(* Logix 5000 project; controller DUNEW2PLC1 vendor 1 type 14 code 221 rev 33.11; software revision 33.00; part 6 of 7 *)
(* tags used below, declared in another part *)
   AbortQueue : BOOL;
   accel_xy : REAL;   // Tangential acceleration of the winding head in xy-plane
   ACTUATOR_POS : DINT;
   ALL_EOT_GOOD : BOOL;
   APA_IS_VERTICAL : BOOL;
   check_tension_stable : BOOL;   // Check if the tension is stable at the setpoint before moving the winding head
   CurIssued : BOOL;
   delay_mid_position : TIMER;
   ENABLE_ACTUATOR : BOOL;
   ERROR_CODE : DINT;
   FRAME_LOC_FT_BTM : BOOL;
   FRAME_LOC_FT_MID : BOOL;
   FRAME_LOC_FT_TOP : BOOL;
   FRAME_LOC_HD_BTM : BOOL;
   FRAME_LOC_HD_MID : BOOL;
   FRAME_LOC_HD_TOP : BOOL;
   gamma : REAL;
   INIT_DONE : BOOL;
   J : REAL;
   LATCH_ACTUATOR_HOMED : BOOL;
   LATCH_ACTUATOR_MID : BOOL;
   LATCH_ACTUATOR_TOP : BOOL;
   latching_in_progress : BOOL;
   MACHINE_SW_STAT : BOOL[32];
   MASTER_Z_GO : BOOL;
   MAX_TOLERABLE_Z : REAL;
   MCCD_X_Y_Axis1 : MOTION_INSTRUCTION;
   MOVE_TYPE : INT;   // 0 = No Move 1 = XY JOG 2 = XY Plane Move 3 = Z JOG 4 = Z Axis Move 5 = Toggle Latch Actuator 6 = Home the Latch Actuator
   NextIssued : BOOL;
   NEXTSTATE : DINT;
   no_apa_collision : BOOL;
   no_latch_collision : BOOL;
   no_supports_collision : BOOL;
   POSITION : REAL[1,2];
   QueueCount : DINT;
   speed_regulator_switch : BOOL;   // This is our "enable safe speed" switch, repurposed to switch the speed regulator
   STATE : DINT;   // CURRENT State Machine State
   STATE_FAULT_FLAGS : DINT;
   STATE_REQUEST : DINT;
   STATE_REQUEST_ACK : DINT;
   STATE_REQUEST_ID : DINT;
   STATE_REQUEST_RESULT : DINT;
   support_collision_window_bttm : BOOL;
   support_collision_window_mid : BOOL;
   support_collision_window_top : BOOL;
   tension : REAL;   // wire tension from load cell (N)
   TENSION_CONTROL_OK : BOOL;
   TENSION_ON_SWITCH : BOOL;
   tension_stable_timer : TIMER;
   v_0 : REAL;
   v_x_max : DINT;
   v_xyz : REAL;   // Velocity of winding head in xyz space
   v_y_max : DINT;
   X_axis : AXIS_CIP_DRIVE;
   X_POSITION : ALIAS FOR POSITION[0,0];
   X_XFER_OK : BOOL;   // If at the head, check head support arms. Same for foot
   X_Y : COORDINATE_SYSTEM;
   XY_ACCELERATION : REAL;   // Maximum positive acceleration for position move.
   XY_DECELERATION : REAL;   // Maximum negative acceleration for position move.
   xy_regulated_acceleration : REAL;
   xy_regulated_deceleration : REAL;
   XY_SPEED : REAL;   // Maximum velocity for position move.
   XY_SPEED_REQ : REAL;   // XY Requested speed copy of XY_Speed to be used for MCLM and MCCD in MoveXY
   xz : COORDINATE_SYSTEM;
   Y_axis : AXIS_CIP_DRIVE;
   Y_POSITION : ALIAS FOR POSITION[0,1];
   Y_XFER_OK : BOOL;
   Z_ACCELERATION : REAL;
   Z_axis : AXIS_CIP_DRIVE;
   Z_DECELLERATION : REAL;
   Z_EXTENDED : BOOL;
   Z_FIXED_LATCHED : BOOL;
   Z_FIXED_PRESENT : BOOL;
   Z_POSITION : REAL;
   Z_RETRACTED : BOOL;
   Z_SPEED : REAL;
   Z_STAGE_LATCHED : BOOL;
   Z_STAGE_PRESENT : BOOL;   // Winding head is on the Z-arm

PROGRAM state_14_hmi_stop   (* main routine main *)
VAR
   hmi_stop_entry_ob : BOOL;
   hmi_stop_entry_sb : BOOL;
   hmi_x_axis_stop : MOTION_INSTRUCTION := (FLAGS := 33554432);
   hmi_xy_stop : MOTION_INSTRUCTION := (FLAGS := 33554432);
   hmi_xz_stop : MOTION_INSTRUCTION := (FLAGS := 33554432);
   hmi_y_axis_stop : MOTION_INSTRUCTION := (FLAGS := 33554432);
   hmi_z_axis_stop : MOTION_INSTRUCTION := (FLAGS := 33554432);
   STATE14_IND : BOOL;
END_VAR

ROUTINE main   (* ladder *)
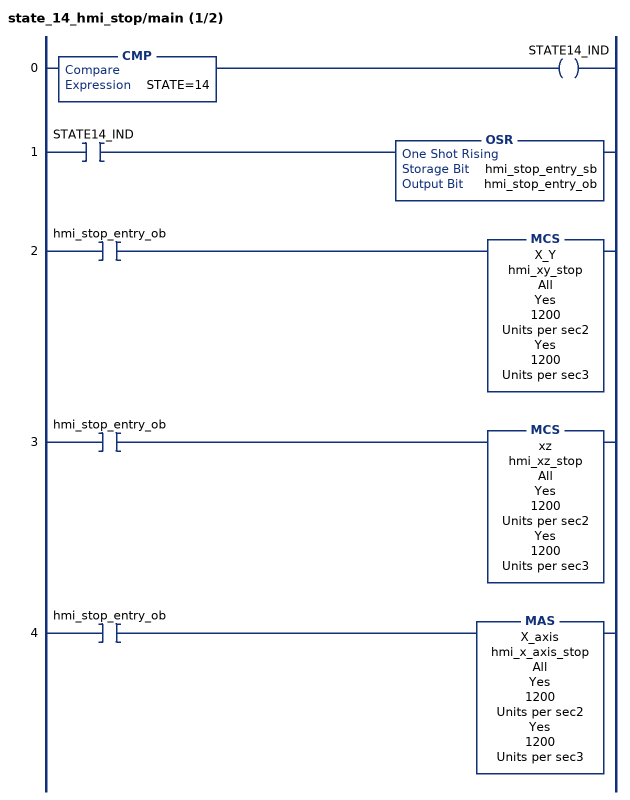
   0: CMP(STATE=14)OTE(STATE14_IND);
   1: XIC(STATE14_IND)OSR(hmi_stop_entry_sb,hmi_stop_entry_ob);
   2: XIC(hmi_stop_entry_ob)MCS(X_Y,hmi_xy_stop,All,Yes,1200,Units per sec2,Yes,1200,Units per sec3);
   3: XIC(hmi_stop_entry_ob)MCS(xz,hmi_xz_stop,All,Yes,1200,Units per sec2,Yes,1200,Units per sec3);
   4: XIC(hmi_stop_entry_ob)MAS(X_axis,hmi_x_axis_stop,All,Yes,1200,Units per sec2,Yes,1200,Units per sec3);
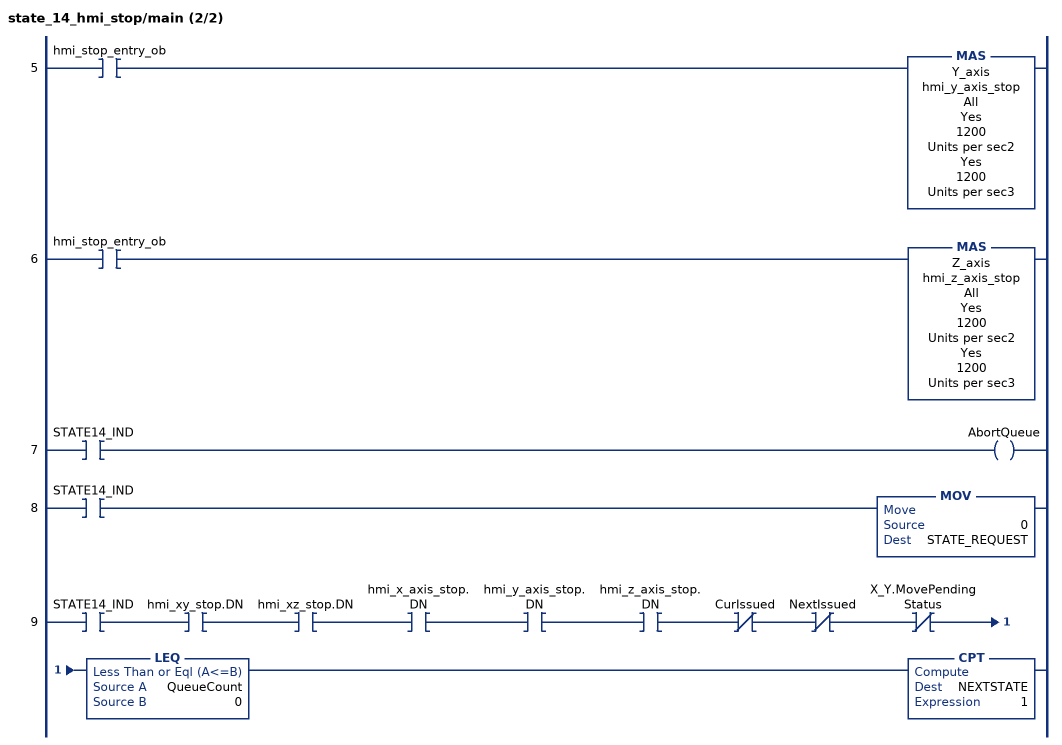
   5: XIC(hmi_stop_entry_ob)MAS(Y_axis,hmi_y_axis_stop,All,Yes,1200,Units per sec2,Yes,1200,Units per sec3);
   6: XIC(hmi_stop_entry_ob)MAS(Z_axis,hmi_z_axis_stop,All,Yes,1200,Units per sec2,Yes,1200,Units per sec3);
   7: XIC(STATE14_IND)OTE(AbortQueue);
   8: XIC(STATE14_IND)MOV(0,STATE_REQUEST);
   9: XIC(STATE14_IND)XIC(hmi_xy_stop.DN)XIC(hmi_xz_stop.DN)XIC(hmi_x_axis_stop.DN)XIC(hmi_y_axis_stop.DN)XIC(hmi_z_axis_stop.DN)XIO(CurIssued)XIO(NextIssued)XIO(X_Y.MovePendingStatus)LEQ(QueueCount,0)CPT(NEXTSTATE,1);
END_ROUTINE
END_PROGRAM

PROGRAM state_1_ready   (* main routine main *)
VAR
   STATE1_IND : BOOL; {access Read Only}
END_VAR

ROUTINE main   (* ladder *)
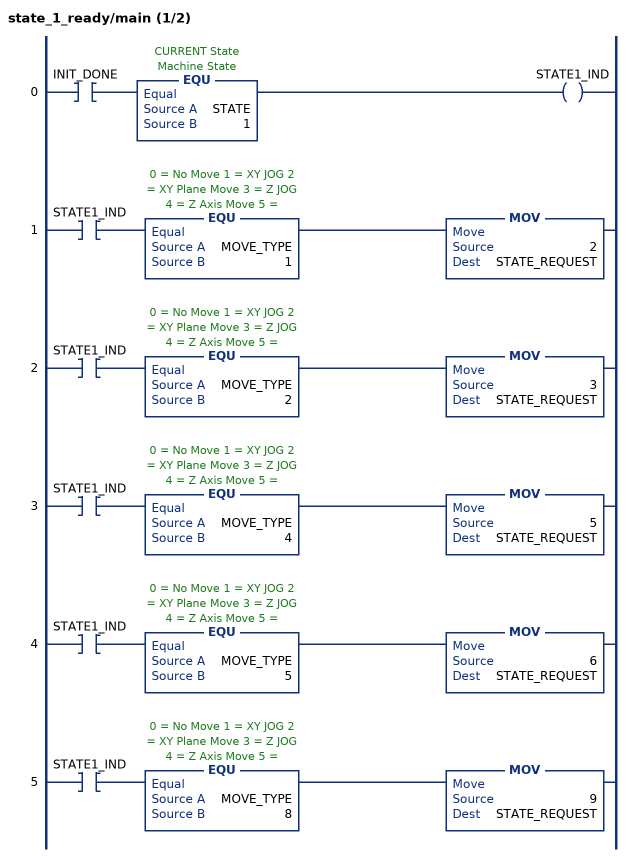
   0: XIC(INIT_DONE)EQU(STATE,1)OTE(STATE1_IND);
   1: XIC(STATE1_IND)EQU(MOVE_TYPE,1)MOV(2,STATE_REQUEST);
   2: XIC(STATE1_IND)EQU(MOVE_TYPE,2)MOV(3,STATE_REQUEST);
   3: XIC(STATE1_IND)EQU(MOVE_TYPE,4)MOV(5,STATE_REQUEST);
   4: XIC(STATE1_IND)EQU(MOVE_TYPE,5)MOV(6,STATE_REQUEST);
   5: XIC(STATE1_IND)EQU(MOVE_TYPE,8)MOV(9,STATE_REQUEST);
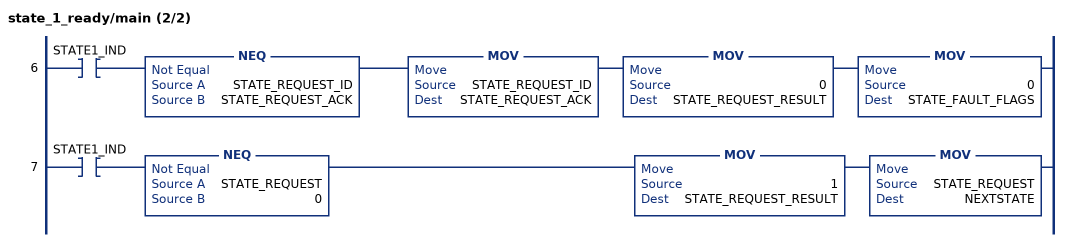
   6: XIC(STATE1_IND)NEQ(STATE_REQUEST_ID,STATE_REQUEST_ACK)MOV(STATE_REQUEST_ID,STATE_REQUEST_ACK)MOV(0,STATE_REQUEST_RESULT)MOV(0,STATE_FAULT_FLAGS);
   7: XIC(STATE1_IND)NEQ(STATE_REQUEST,0)MOV(1,STATE_REQUEST_RESULT)MOV(STATE_REQUEST,NEXTSTATE);
END_ROUTINE
END_PROGRAM

PROGRAM state_3_move_xy   (* main routine main *)
VAR
   auto_edge_0_sb : BOOL;
   d_raw : REAL;
   dx : REAL := 443.4121;
   dy : REAL := 196.90817;
   eot_triggered : BOOL;
   k : REAL := 1.8605716;
   main_xy_move : MOTION_INSTRUCTION;
   main_xy_move_completed : BOOL;
   main_xy_move_completed_sb : BOOL;
   max_integral : DINT := 1000;
   min_integral : DINT := -1000;
   min_regulated_speed : DINT := 100;
   move_xy_entry_ob : BOOL;
   move_xy_entry_sb : BOOL;
   near_ending : BOOL := 1;   // True if distance to xy-move target is less than the required stopping distance
   regulated_speed : REAL := 902.6882;
   regulator_loop_timer : TIMER := (PRE := 1, EN := 1, TT := 1);
   speed_regulator_off_ob : BOOL;
   speed_regulator_off_sb : BOOL := 1;
   speed_tension_setpoint : REAL := 8.5;
   starting_x : REAL := 6726.988;
   starting_y : REAL := 112.5774;
   STATE3_IND : BOOL; {access Read Only}
   stopping_distance : REAL := 37.499752;   // Calculate the distance required to perform a jerk-limited stop at the gurrent jerk, acceleration, and speed
   stopping_ratio : REAL := 9.108512e-05;
   trigger_xy_move : BOOL;
   v_max : REAL := 902.6882;
   x_axis_mso : MOTION_INSTRUCTION := (FLAGS := 536870912, DN := 1);
   x_dist_to_target : REAL := 0.00048828125;
   x_time : REAL := 1.8605716;
   xy_accel_jerk : DINT := 2000;
   xy_axes_servoed_on_ob : BOOL;
   xy_axes_servoed_on_sb : BOOL := 1;
   xy_d_alpha : REAL := 1.0;
   xy_d_dt : DINT := 50;
   xy_d_term : REAL;
   xy_d_term_prev : REAL;
   xy_d_timer : TIMER := (PRE := 50, ACC := 3, EN := 1, TT := 1);
   xy_decel_jerk : DINT := 2000;
   xy_default_speed : DINT;
   xy_dist_to_target : REAL := 0.00049208116;
   xy_dt : DINT := 1;
   xy_eot_stop_control : MOTION_INSTRUCTION := (FLAGS := 570425344, DN := 1);
   xy_error : REAL := 2.1404376;
   xy_error_prev : REAL := 2.1455598;
   xy_i_term : REAL := 902.72687;
   xy_kd : REAL;
   xy_ki : REAL := 300.0;
   xy_kp : REAL;
   xy_move_error_ob : BOOL;
   xy_move_error_sb : BOOL;
   xy_move_trigger_sb : BOOL;
   xy_p_term : REAL;
   xy_pre_move : BOOL;
   xy_regulated_accel_jerk : DINT := 800;
   y_axis_mso : MOTION_INSTRUCTION := (FLAGS := 536870912, DN := 1);
   y_dist_to_target : REAL := -0.00015258789;
   y_time : REAL := 3.0471056;
   z_axis_mso : MOTION_INSTRUCTION;
   z_axis_pre_xy_retract : MOTION_INSTRUCTION := (FLAGS := 671088640, DN := 1, PC := 1);
END_VAR

ROUTINE main   (* ladder *)
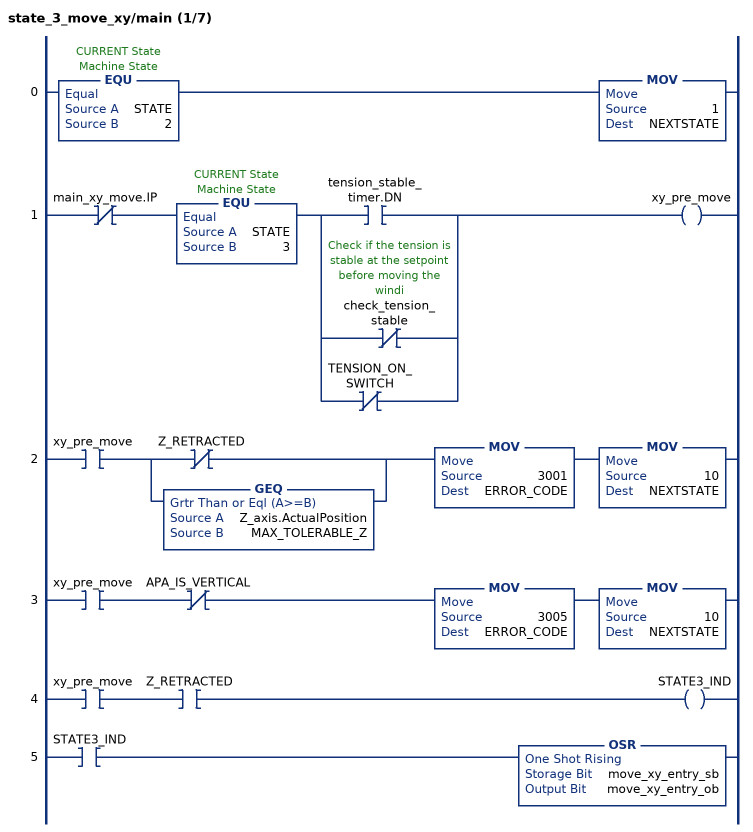
   0: EQU(STATE,2)MOV(1,NEXTSTATE);
   1: XIO(main_xy_move.IP)EQU(STATE,3)[XIC(tension_stable_timer.DN) ,XIO(check_tension_stable) ,XIO(TENSION_ON_SWITCH) ]OTE(xy_pre_move);
   2: XIC(xy_pre_move)[XIO(Z_RETRACTED) ,GEQ(Z_axis.ActualPosition,MAX_TOLERABLE_Z) ]MOV(3001,ERROR_CODE)MOV(10,NEXTSTATE);
   3: XIC(xy_pre_move)XIO(APA_IS_VERTICAL)MOV(3005,ERROR_CODE)MOV(10,NEXTSTATE);
   4: XIC(xy_pre_move)XIC(Z_RETRACTED)OTE(STATE3_IND);
   5: XIC(STATE3_IND)OSR(move_xy_entry_sb,move_xy_entry_ob);
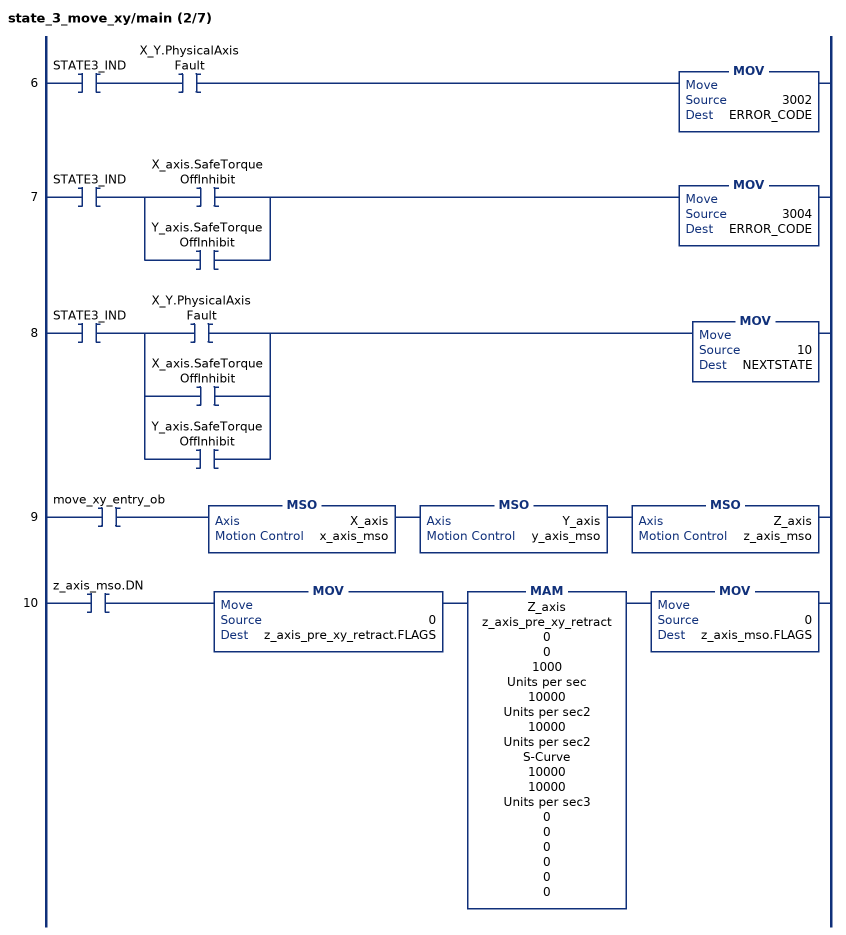
   6: XIC(STATE3_IND)XIC(X_Y.PhysicalAxisFault)MOV(3002,ERROR_CODE);
   7: XIC(STATE3_IND)[XIC(X_axis.SafeTorqueOffInhibit) ,XIC(Y_axis.SafeTorqueOffInhibit) ]MOV(3004,ERROR_CODE);
   8: XIC(STATE3_IND)[XIC(X_Y.PhysicalAxisFault) ,XIC(X_axis.SafeTorqueOffInhibit) ,XIC(Y_axis.SafeTorqueOffInhibit) ]MOV(10,NEXTSTATE);
   9: XIC(move_xy_entry_ob)MSO(X_axis,x_axis_mso)MSO(Y_axis,y_axis_mso)MSO(Z_axis,z_axis_mso);
   10: XIC(z_axis_mso.DN)MOV(0,z_axis_pre_xy_retract.FLAGS)MAM(Z_axis,z_axis_pre_xy_retract,0,0,1000,Units per sec,10000,Units per sec2,10000,Units per sec2,S-Curve,10000,10000,Units per sec3,0,0,0,0,0,0)MOV(0,z_axis_mso.FLAGS);
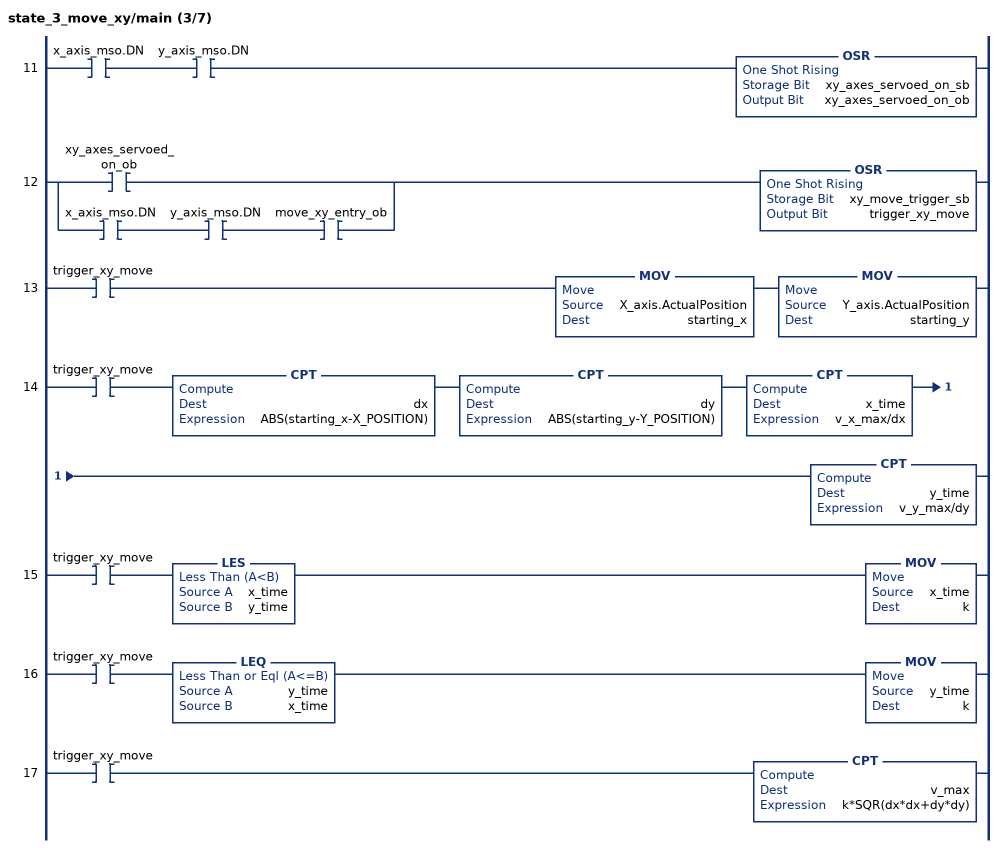
   11: XIC(x_axis_mso.DN)XIC(y_axis_mso.DN)OSR(xy_axes_servoed_on_sb,xy_axes_servoed_on_ob);
   12: [XIC(xy_axes_servoed_on_ob) ,XIC(x_axis_mso.DN) XIC(y_axis_mso.DN) XIC(move_xy_entry_ob) ]OSR(xy_move_trigger_sb,trigger_xy_move);
   13: XIC(trigger_xy_move)MOV(X_axis.ActualPosition,starting_x)MOV(Y_axis.ActualPosition,starting_y);
   14: XIC(trigger_xy_move)CPT(dx,ABS(starting_x-X_POSITION))CPT(dy,ABS(starting_y-Y_POSITION))CPT(x_time,v_x_max/dx)CPT(y_time,v_y_max/dy);
   15: XIC(trigger_xy_move)LES(x_time,y_time)MOV(x_time,k);
   16: XIC(trigger_xy_move)LEQ(y_time,x_time)MOV(y_time,k);
   17: XIC(trigger_xy_move)CPT(v_max,k*SQR(dx*dx+dy*dy));
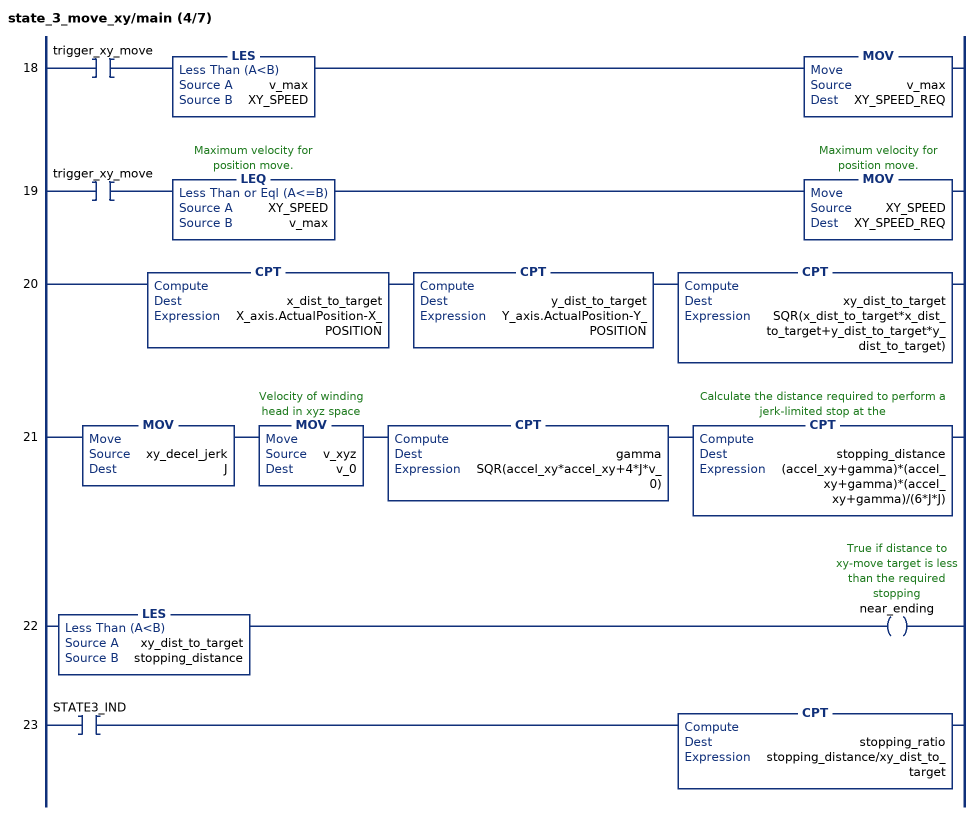
   18: XIC(trigger_xy_move)LES(v_max,XY_SPEED)MOV(v_max,XY_SPEED_REQ);
   19: XIC(trigger_xy_move)LEQ(XY_SPEED,v_max)MOV(XY_SPEED,XY_SPEED_REQ);
   20: CPT(x_dist_to_target,X_axis.ActualPosition-X_POSITION)CPT(y_dist_to_target,Y_axis.ActualPosition-Y_POSITION)CPT(xy_dist_to_target,SQR(x_dist_to_target*x_dist_to_target+y_dist_to_target*y_dist_to_target));
   21: MOV(xy_decel_jerk,J)MOV(v_xyz,v_0)CPT(gamma,SQR(accel_xy*accel_xy+4*J*v_0))CPT(stopping_distance,(accel_xy+gamma)*(accel_xy+gamma)*(accel_xy+gamma)/(6*J*J));
   22: LES(xy_dist_to_target,stopping_distance)OTE(near_ending);
   23: XIC(STATE3_IND)CPT(stopping_ratio,stopping_distance/xy_dist_to_target);
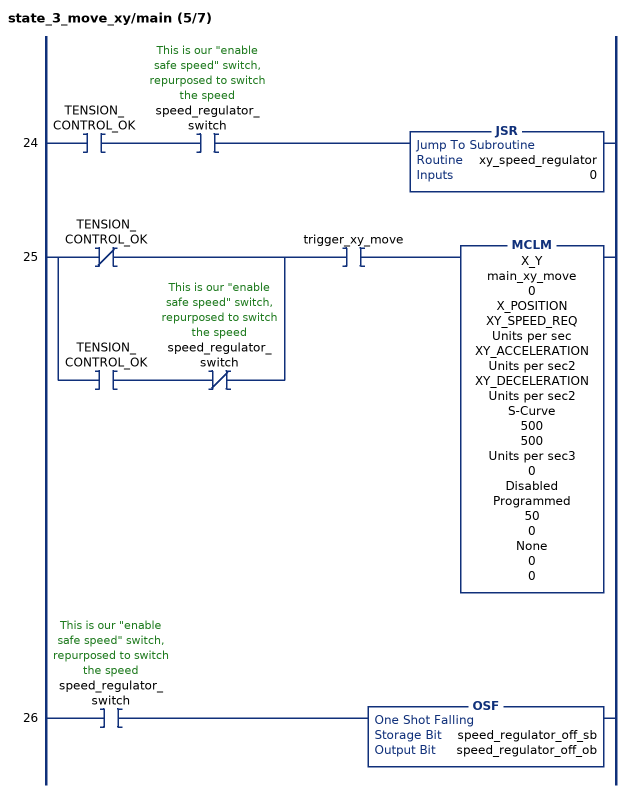
   24: XIC(TENSION_CONTROL_OK)XIC(speed_regulator_switch)JSR(xy_speed_regulator,0);
   25: [XIO(TENSION_CONTROL_OK) ,XIC(TENSION_CONTROL_OK) XIO(speed_regulator_switch) ]XIC(trigger_xy_move)MCLM(X_Y,main_xy_move,0,X_POSITION,XY_SPEED_REQ,Units per sec,XY_ACCELERATION,Units per sec2,XY_DECELERATION,Units per sec2,S-Curve,500,500,Units per sec3,0,Disabled,Programmed,50,0,None,0,0);
   26: XIC(speed_regulator_switch)OSF(speed_regulator_off_sb,speed_regulator_off_ob);
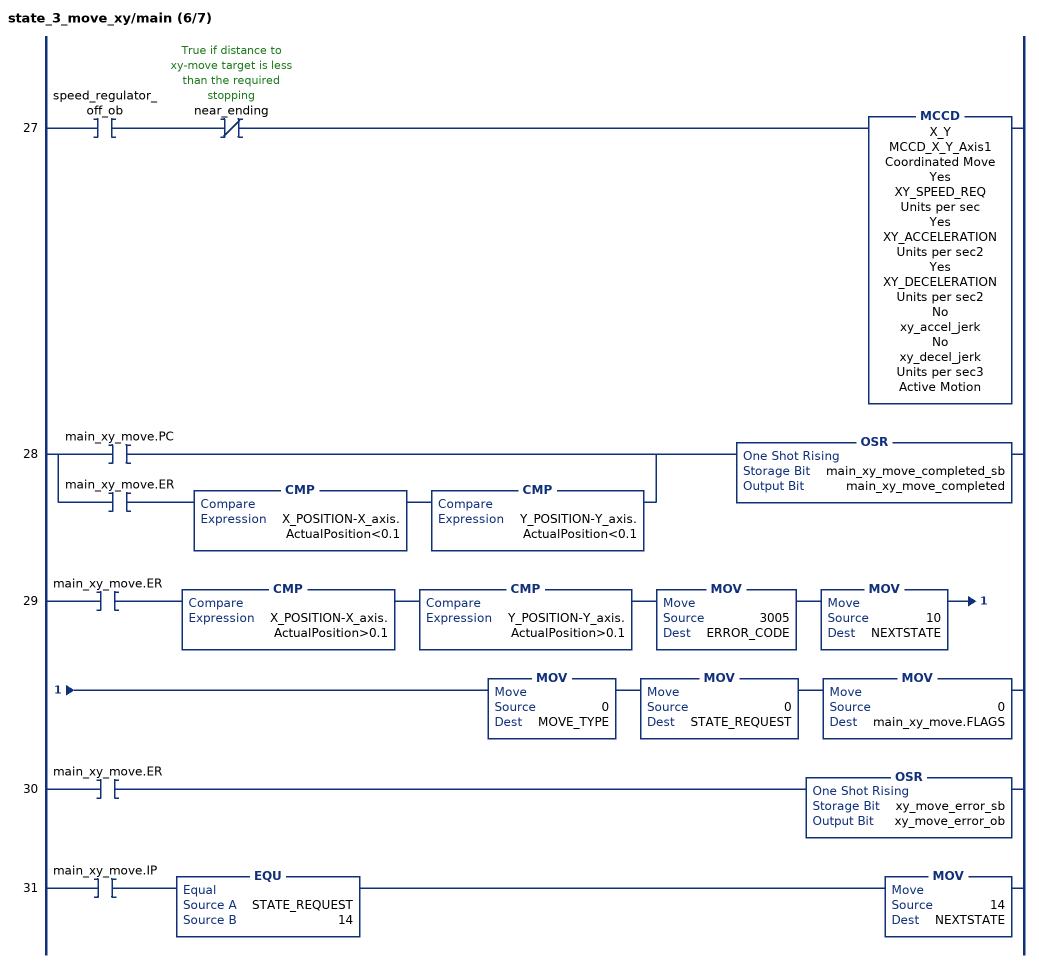
   27: XIC(speed_regulator_off_ob)XIO(near_ending)MCCD(X_Y,MCCD_X_Y_Axis1,Coordinated Move,Yes,XY_SPEED_REQ,Units per sec,Yes,XY_ACCELERATION,Units per sec2,Yes,XY_DECELERATION,Units per sec2,No,xy_accel_jerk,No,xy_decel_jerk,Units per sec3,Active Motion);
   28: [XIC(main_xy_move.PC) ,XIC(main_xy_move.ER) CMP(X_POSITION-X_axis.ActualPosition<0.1) CMP(Y_POSITION-Y_axis.ActualPosition<0.1) ]OSR(main_xy_move_completed_sb,main_xy_move_completed);
   29: XIC(main_xy_move.ER)CMP(X_POSITION-X_axis.ActualPosition>0.1)CMP(Y_POSITION-Y_axis.ActualPosition>0.1)MOV(3005,ERROR_CODE)MOV(10,NEXTSTATE)MOV(0,MOVE_TYPE)MOV(0,STATE_REQUEST)MOV(0,main_xy_move.FLAGS);
   30: XIC(main_xy_move.ER)OSR(xy_move_error_sb,xy_move_error_ob);
   31: XIC(main_xy_move.IP)EQU(STATE_REQUEST,14)MOV(14,NEXTSTATE);
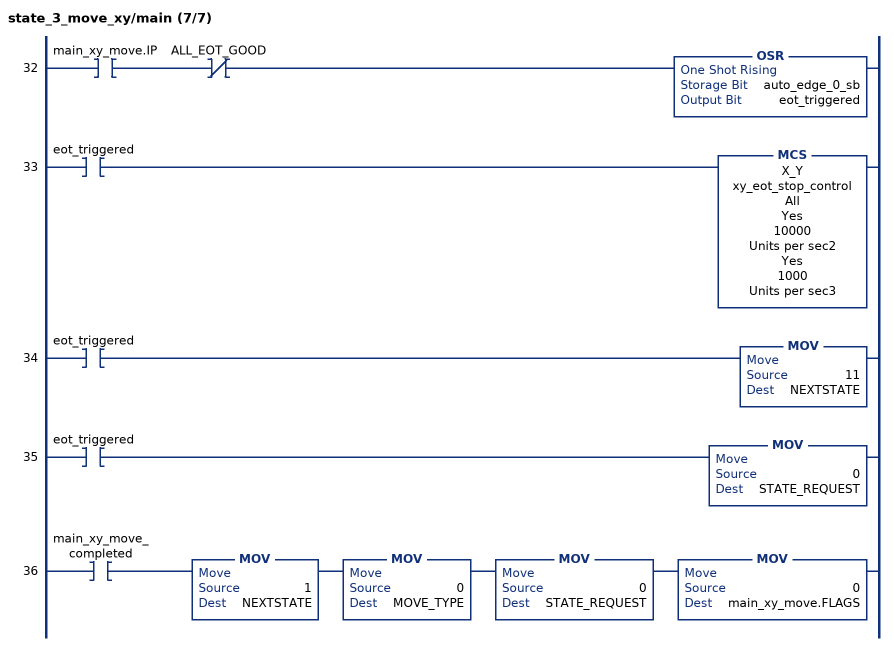
   32: XIC(main_xy_move.IP)XIO(ALL_EOT_GOOD)OSR(auto_edge_0_sb,eot_triggered);
   33: XIC(eot_triggered)MCS(X_Y,xy_eot_stop_control,All,Yes,10000,Units per sec2,Yes,1000,Units per sec3);
   34: XIC(eot_triggered)MOV(11,NEXTSTATE);
   35: XIC(eot_triggered)MOV(0,STATE_REQUEST);
   36: XIC(main_xy_move_completed)MOV(1,NEXTSTATE)MOV(0,MOVE_TYPE)MOV(0,STATE_REQUEST)MOV(0,main_xy_move.FLAGS);
END_ROUTINE

ROUTINE xy_speed_regulator   (* ladder *)
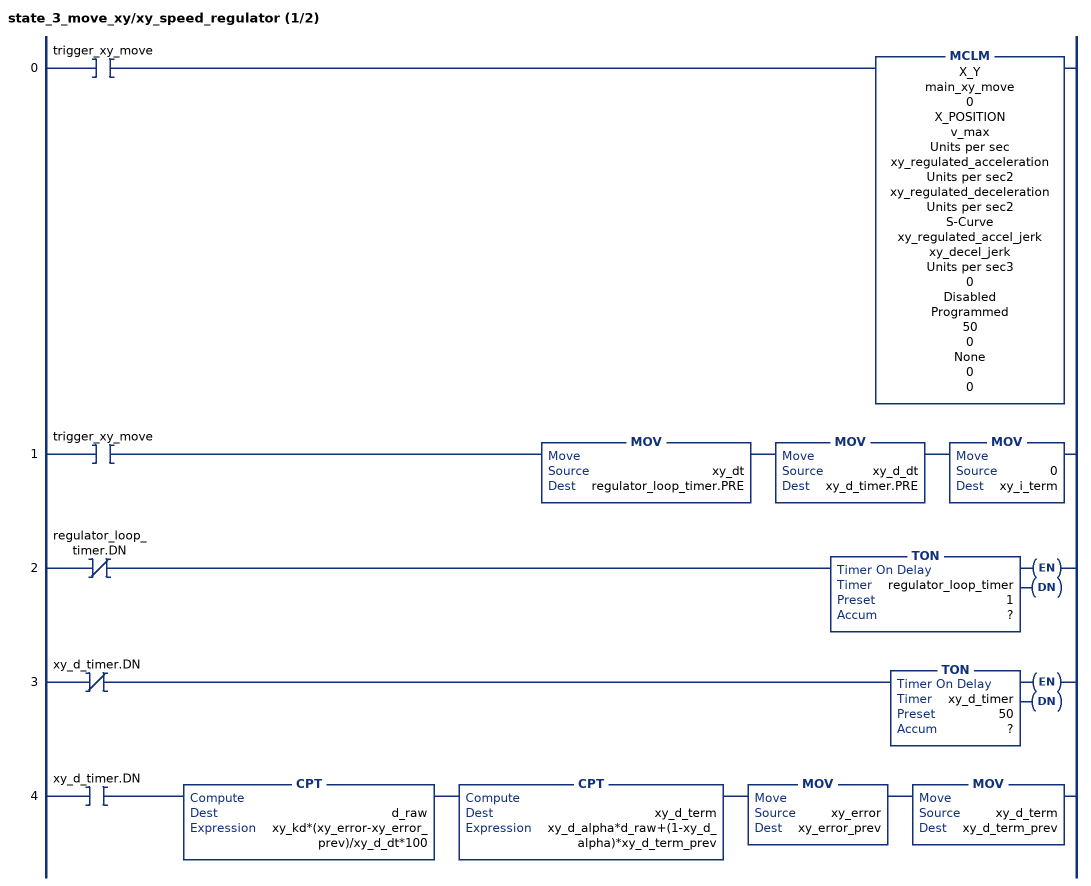
   0: XIC(trigger_xy_move)MCLM(X_Y,main_xy_move,0,X_POSITION,v_max,Units per sec,xy_regulated_acceleration,Units per sec2,xy_regulated_deceleration,Units per sec2,S-Curve,xy_regulated_accel_jerk,xy_decel_jerk,Units per sec3,0,Disabled,Programmed,50,0,None,0,0);
   1: XIC(trigger_xy_move)MOV(xy_dt,regulator_loop_timer.PRE)MOV(xy_d_dt,xy_d_timer.PRE)MOV(0,xy_i_term);
   2: XIO(regulator_loop_timer.DN)TON(regulator_loop_timer,?,?);
   3: XIO(xy_d_timer.DN)TON(xy_d_timer,?,?);
   4: XIC(xy_d_timer.DN)CPT(d_raw,xy_kd*(xy_error-xy_error_prev)/xy_d_dt*100)CPT(xy_d_term,xy_d_alpha*d_raw+(1-xy_d_alpha)*xy_d_term_prev)MOV(xy_error,xy_error_prev)MOV(xy_d_term,xy_d_term_prev);
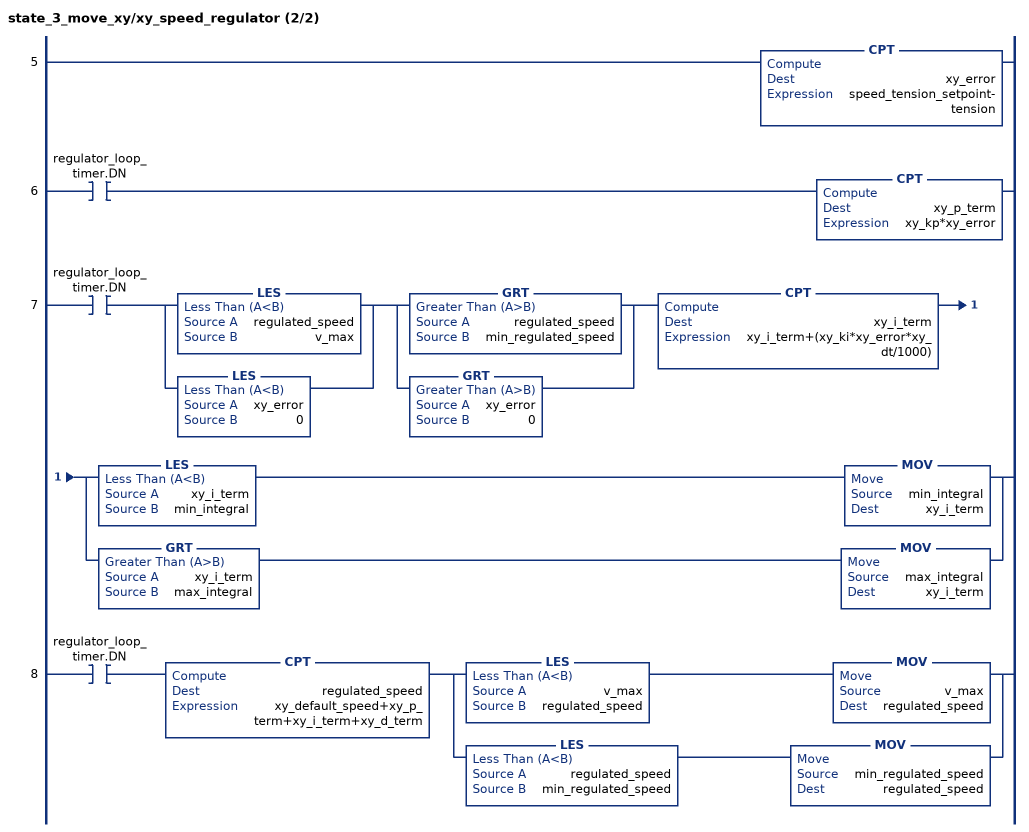
   5: CPT(xy_error,speed_tension_setpoint-tension);
   6: XIC(regulator_loop_timer.DN)CPT(xy_p_term,xy_kp*xy_error);
   7: XIC(regulator_loop_timer.DN)[LES(regulated_speed,v_max) ,LES(xy_error,0) ][GRT(regulated_speed,min_regulated_speed) ,GRT(xy_error,0) ]CPT(xy_i_term,xy_i_term+(xy_ki*xy_error*xy_dt/1000))[LES(xy_i_term,min_integral) MOV(min_integral,xy_i_term) ,GRT(xy_i_term,max_integral) MOV(max_integral,xy_i_term) ];
   8: XIC(regulator_loop_timer.DN)CPT(regulated_speed,xy_default_speed+xy_p_term+xy_i_term+xy_d_term)[LES(v_max,regulated_speed) MOV(v_max,regulated_speed) ,LES(regulated_speed,min_regulated_speed) MOV(min_regulated_speed,regulated_speed) ];
END_ROUTINE
END_PROGRAM

PROGRAM state_5_move_z   (* main routine main *)
VAR
   eot_stop : MOTION_INSTRUCTION := (FLAGS := 33554432);
   oneshotob : BOOL[32]; {access Read Only}
   STATE5_IND : BOOL := 1; {access Read Only}
   z_accel_jerk : DINT := 500;
   z_axis_fast_move : MOTION_INSTRUCTION := (FLAGS := -1543503870, EN := 1, DN := 1, IP := 1, DECEL := 1);
   z_axis_main_move : MOTION_INSTRUCTION;
   z_axis_mso : MOTION_INSTRUCTION;
   z_decel_jerk : DINT := 1000;
   z_move_success : BOOL;
END_VAR

ROUTINE main   (* ladder *)
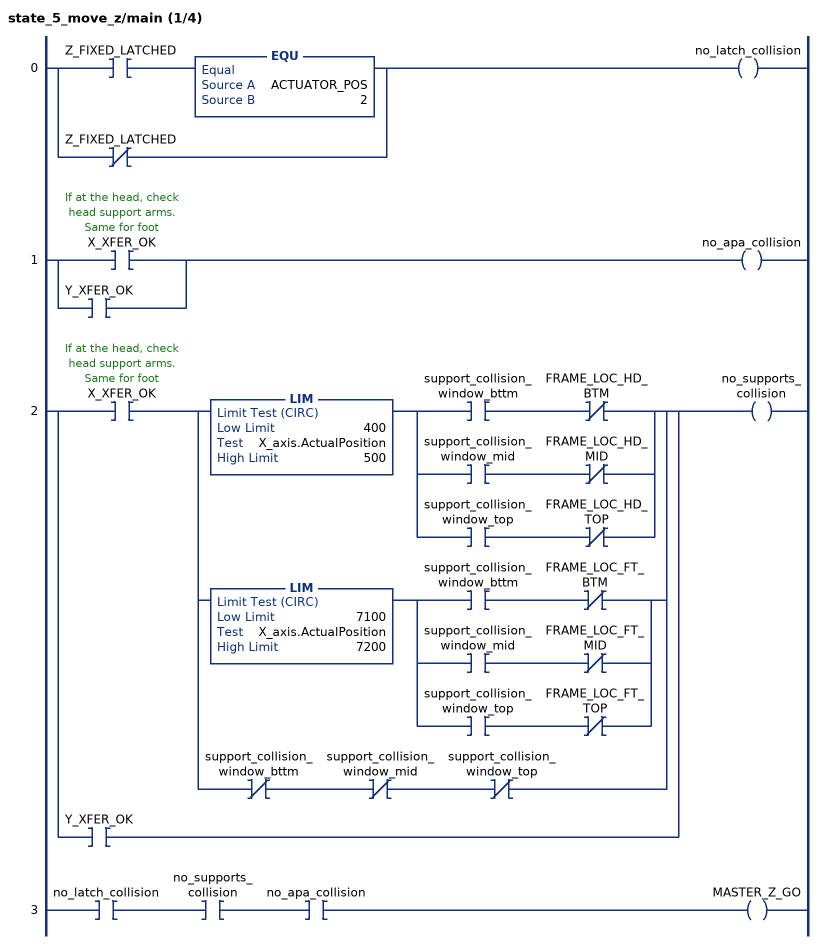
   0: [XIC(Z_FIXED_LATCHED) EQU(ACTUATOR_POS,2) ,XIO(Z_FIXED_LATCHED) ]OTE(no_latch_collision);
   1: [XIC(X_XFER_OK) ,XIC(Y_XFER_OK) ]OTE(no_apa_collision);
   2: [XIC(X_XFER_OK) [LIM(400,X_axis.ActualPosition,500) [XIC(support_collision_window_bttm) XIO(FRAME_LOC_HD_BTM) ,XIC(support_collision_window_mid) XIO(FRAME_LOC_HD_MID) ,XIC(support_collision_window_top) XIO(FRAME_LOC_HD_TOP) ] ,LIM(7100,X_axis.ActualPosition,7200) [XIC(support_collision_window_bttm) XIO(FRAME_LOC_FT_BTM) ,XIC(support_collision_window_mid) XIO(FRAME_LOC_FT_MID) ,XIC(support_collision_window_top) XIO(FRAME_LOC_FT_TOP) ] ,XIO(support_collision_window_bttm) XIO(support_collision_window_mid) XIO(support_collision_window_top) ] ,XIC(Y_XFER_OK) ]OTE(no_supports_collision);
   3: XIC(no_latch_collision)XIC(no_supports_collision)XIC(no_apa_collision)OTE(MASTER_Z_GO);
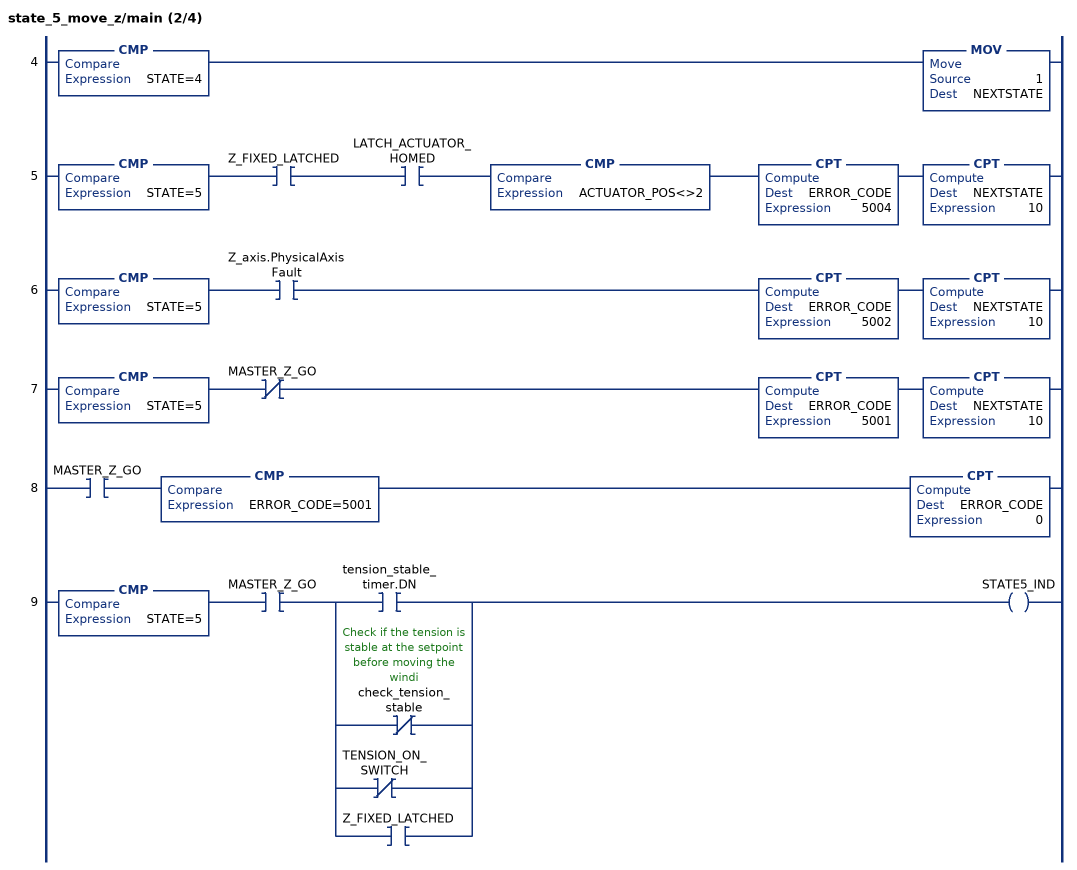
   4: CMP(STATE=4)MOV(1,NEXTSTATE);
   5: CMP(STATE=5)XIC(Z_FIXED_LATCHED)XIC(LATCH_ACTUATOR_HOMED)CMP(ACTUATOR_POS<>2)CPT(ERROR_CODE,5004)CPT(NEXTSTATE,10);
   6: CMP(STATE=5)XIC(Z_axis.PhysicalAxisFault)CPT(ERROR_CODE,5002)CPT(NEXTSTATE,10);
   7: CMP(STATE=5)XIO(MASTER_Z_GO)CPT(ERROR_CODE,5001)CPT(NEXTSTATE,10);
   8: XIC(MASTER_Z_GO)CMP(ERROR_CODE=5001)CPT(ERROR_CODE,0);
   9: CMP(STATE=5)XIC(MASTER_Z_GO)[XIC(tension_stable_timer.DN) ,XIO(check_tension_stable) ,XIO(TENSION_ON_SWITCH) ,XIC(Z_FIXED_LATCHED) ]OTE(STATE5_IND);
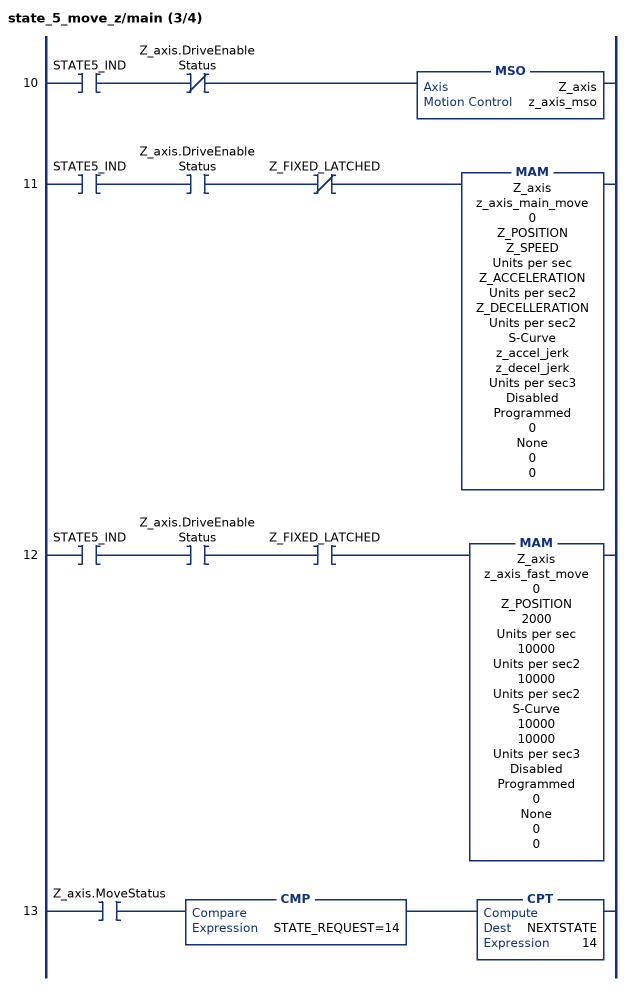
   10: XIC(STATE5_IND)XIO(Z_axis.DriveEnableStatus)MSO(Z_axis,z_axis_mso);
   11: XIC(STATE5_IND)XIC(Z_axis.DriveEnableStatus)XIO(Z_FIXED_LATCHED)MAM(Z_axis,z_axis_main_move,0,Z_POSITION,Z_SPEED,Units per sec,Z_ACCELERATION,Units per sec2,Z_DECELLERATION,Units per sec2,S-Curve,z_accel_jerk,z_decel_jerk,Units per sec3,Disabled,Programmed,0,None,0,0);
   12: XIC(STATE5_IND)XIC(Z_axis.DriveEnableStatus)XIC(Z_FIXED_LATCHED)MAM(Z_axis,z_axis_fast_move,0,Z_POSITION,2000,Units per sec,10000,Units per sec2,10000,Units per sec2,S-Curve,10000,10000,Units per sec3,Disabled,Programmed,0,None,0,0);
   13: XIC(Z_axis.MoveStatus)CMP(STATE_REQUEST=14)CPT(NEXTSTATE,14);
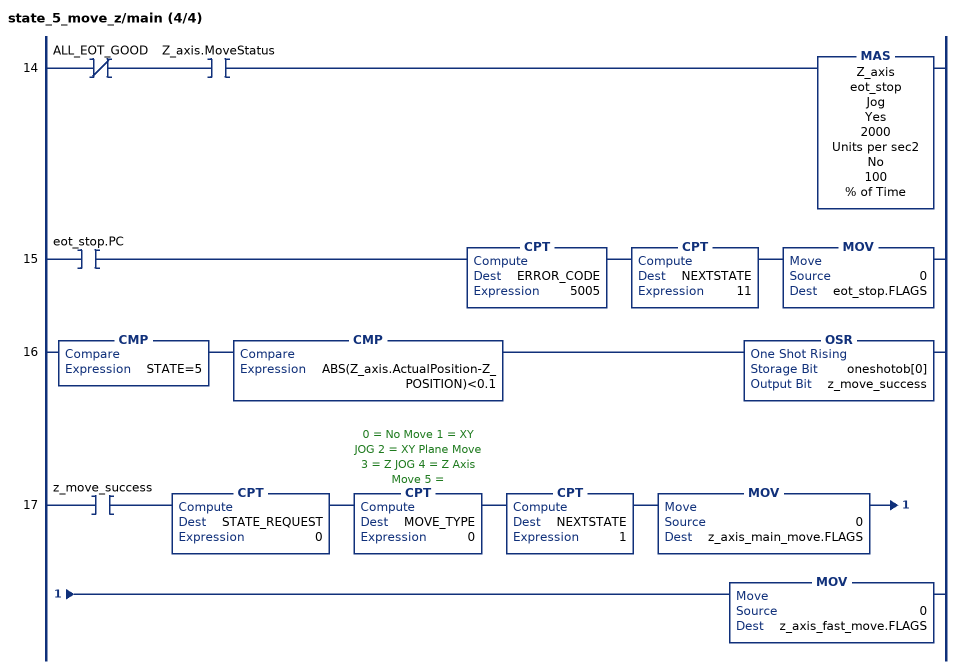
   14: XIO(ALL_EOT_GOOD)XIC(Z_axis.MoveStatus)MAS(Z_axis,eot_stop,Jog,Yes,2000,Units per sec2,No,100,% of Time);
   15: XIC(eot_stop.PC)CPT(ERROR_CODE,5005)CPT(NEXTSTATE,11)MOV(0,eot_stop.FLAGS);
   16: CMP(STATE=5)CMP(ABS(Z_axis.ActualPosition-Z_POSITION)<0.1)OSR(oneshotob[0],z_move_success);
   17: XIC(z_move_success)CPT(STATE_REQUEST,0)CPT(MOVE_TYPE,0)CPT(NEXTSTATE,1)MOV(0,z_axis_main_move.FLAGS)MOV(0,z_axis_fast_move.FLAGS);
END_ROUTINE
END_PROGRAM

PROGRAM state_6_latch   (* main routine main *)
VAR
   delay_stage_latched : TIMER := (PRE := 150);
   head_between_stage_and_fixed : BOOL;
   latch_in_free_space : BOOL;
   Latching_pulse_duration : TIMER := (PRE := 25); {access Read Only}
   Latching_pulse_interval : TIMER := (PRE := 300);
   latching_rising_edge : BOOL;
   latching_signal : BOOL;
   latching_storage_bit : BOOL;
   LatchingTimeoutCounter : COUNTER := (PRE := 20);   // When you enter state 6 or 7, start counting seconds
   manual_toggle_latch : BOOL;
   one_second_timer : TIMER := (PRE := 1000);
   PREV_ACT_POS : DINT := 3; {access Read Only}   // Store the previous actuator position
END_VAR

ROUTINE main   (* ladder *)
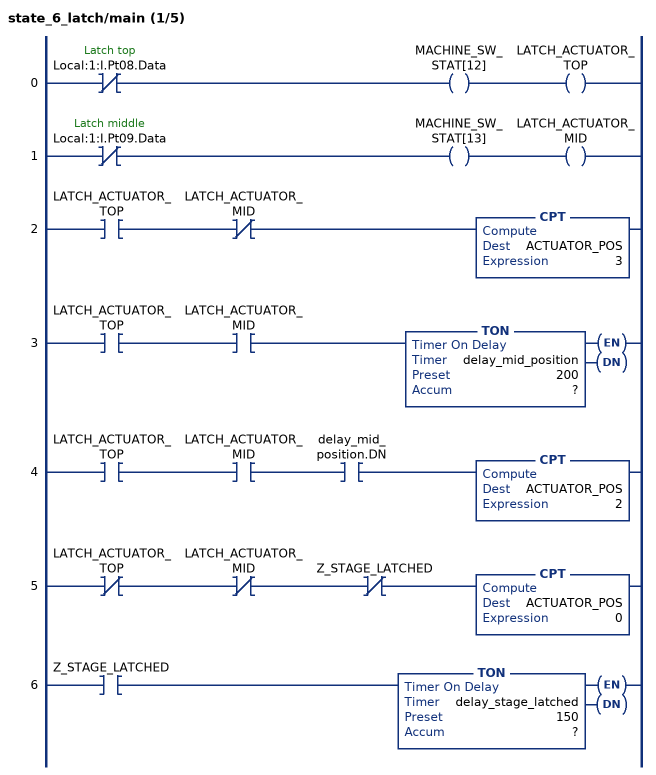
   0: XIO(Local:1:I.Pt08.Data)OTE(MACHINE_SW_STAT[12])OTE(LATCH_ACTUATOR_TOP);
   1: XIO(Local:1:I.Pt09.Data)OTE(MACHINE_SW_STAT[13])OTE(LATCH_ACTUATOR_MID);
   2: XIC(LATCH_ACTUATOR_TOP)XIO(LATCH_ACTUATOR_MID)CPT(ACTUATOR_POS,3);
   3: XIC(LATCH_ACTUATOR_TOP)XIC(LATCH_ACTUATOR_MID)TON(delay_mid_position,?,?);
   4: XIC(LATCH_ACTUATOR_TOP)XIC(LATCH_ACTUATOR_MID)XIC(delay_mid_position.DN)CPT(ACTUATOR_POS,2);
   5: XIO(LATCH_ACTUATOR_TOP)XIO(LATCH_ACTUATOR_MID)XIO(Z_STAGE_LATCHED)CPT(ACTUATOR_POS,0);
   6: XIC(Z_STAGE_LATCHED)TON(delay_stage_latched,?,?);
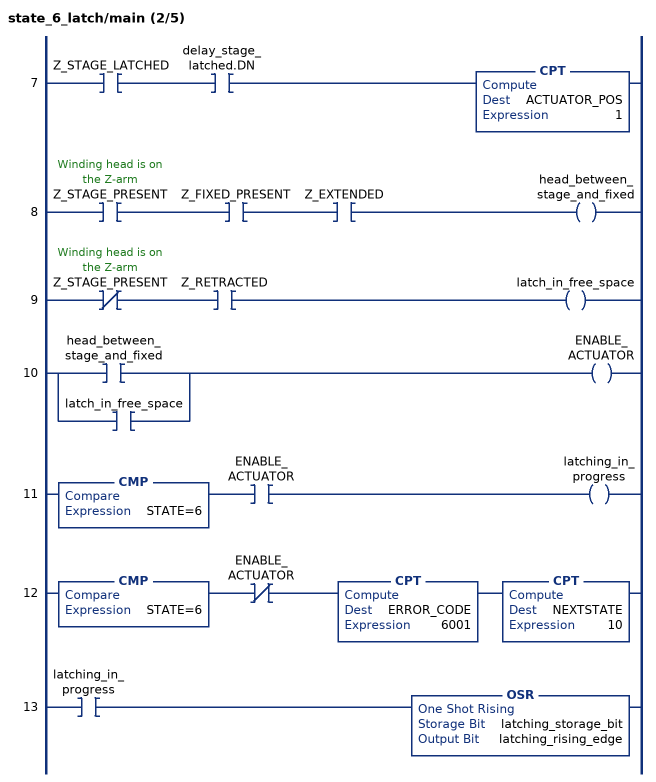
   7: XIC(Z_STAGE_LATCHED)XIC(delay_stage_latched.DN)CPT(ACTUATOR_POS,1);
   8: XIC(Z_STAGE_PRESENT)XIC(Z_FIXED_PRESENT)XIC(Z_EXTENDED)OTE(head_between_stage_and_fixed);
   9: XIO(Z_STAGE_PRESENT)XIC(Z_RETRACTED)OTE(latch_in_free_space);
   10: [XIC(head_between_stage_and_fixed) ,XIC(latch_in_free_space) ]OTE(ENABLE_ACTUATOR);
   11: CMP(STATE=6)XIC(ENABLE_ACTUATOR)OTE(latching_in_progress);
   12: CMP(STATE=6)XIO(ENABLE_ACTUATOR)CPT(ERROR_CODE,6001)CPT(NEXTSTATE,10);
   13: XIC(latching_in_progress)OSR(latching_storage_bit,latching_rising_edge);
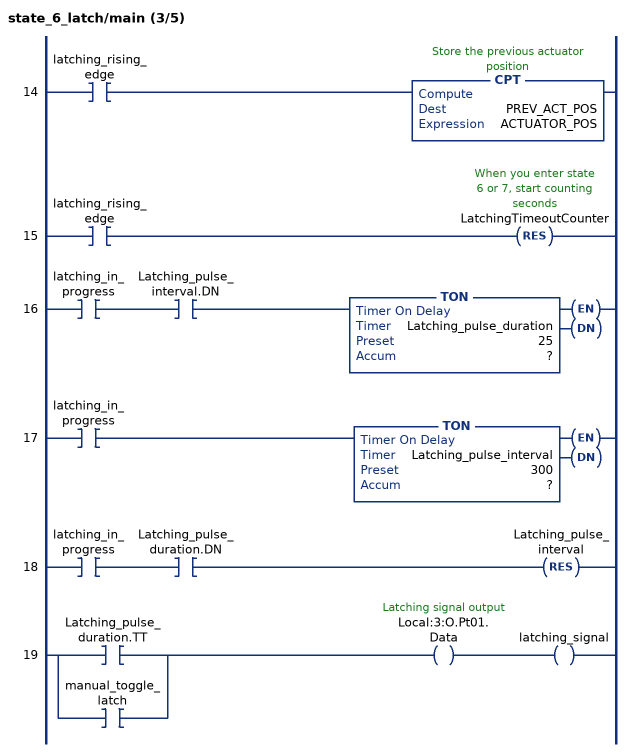
   14: XIC(latching_rising_edge)CPT(PREV_ACT_POS,ACTUATOR_POS);
   15: XIC(latching_rising_edge)RES(LatchingTimeoutCounter);
   16: XIC(latching_in_progress)XIC(Latching_pulse_interval.DN)TON(Latching_pulse_duration,?,?);
   17: XIC(latching_in_progress)TON(Latching_pulse_interval,?,?);
   18: XIC(latching_in_progress)XIC(Latching_pulse_duration.DN)RES(Latching_pulse_interval);
   19: [XIC(Latching_pulse_duration.TT) ,XIC(manual_toggle_latch) ]OTE(Local:3:O.Pt01.Data)OTE(latching_signal);
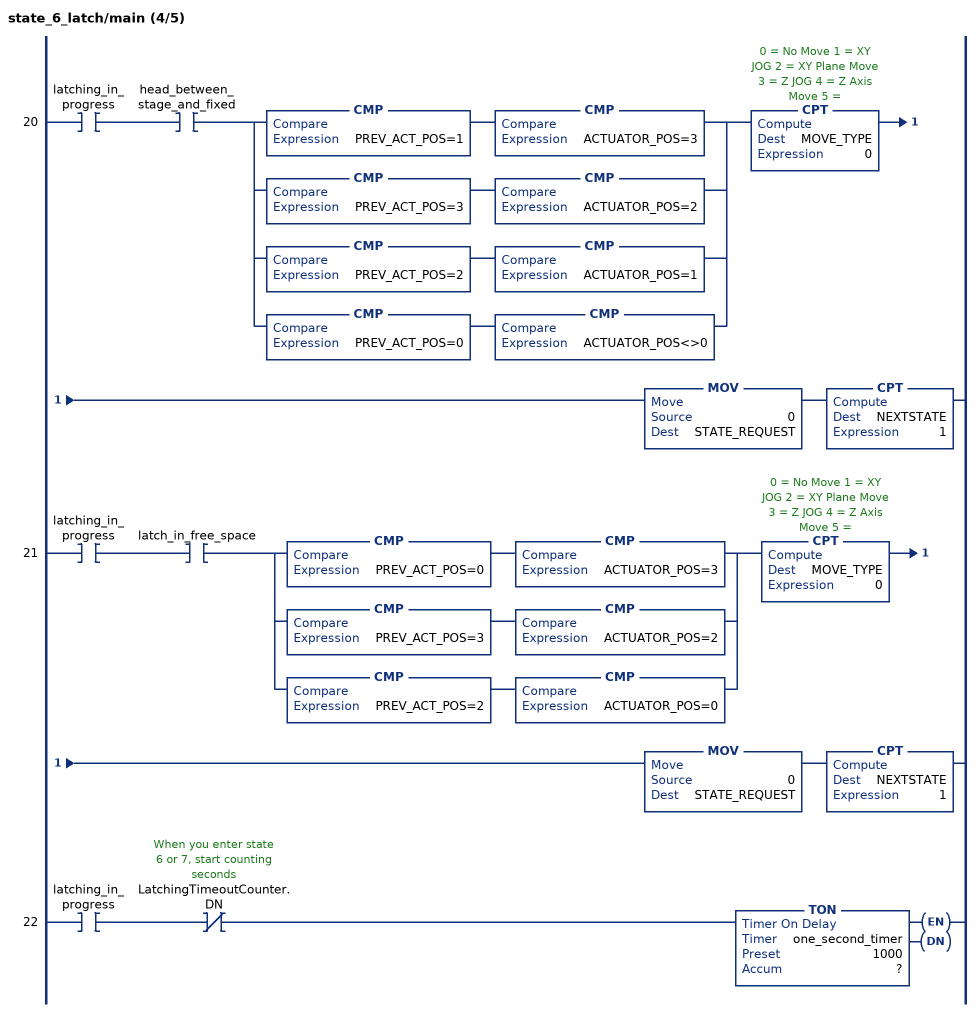
   20: XIC(latching_in_progress)XIC(head_between_stage_and_fixed)[CMP(PREV_ACT_POS=1) CMP(ACTUATOR_POS=3) ,CMP(PREV_ACT_POS=3) CMP(ACTUATOR_POS=2) ,CMP(PREV_ACT_POS=2) CMP(ACTUATOR_POS=1) ,CMP(PREV_ACT_POS=0) CMP(ACTUATOR_POS<>0) ]CPT(MOVE_TYPE,0)MOV(0,STATE_REQUEST)CPT(NEXTSTATE,1);
   21: XIC(latching_in_progress)XIC(latch_in_free_space)[CMP(PREV_ACT_POS=0) CMP(ACTUATOR_POS=3) ,CMP(PREV_ACT_POS=3) CMP(ACTUATOR_POS=2) ,CMP(PREV_ACT_POS=2) CMP(ACTUATOR_POS=0) ]CPT(MOVE_TYPE,0)MOV(0,STATE_REQUEST)CPT(NEXTSTATE,1);
   22: XIC(latching_in_progress)XIO(LatchingTimeoutCounter.DN)TON(one_second_timer,?,?);
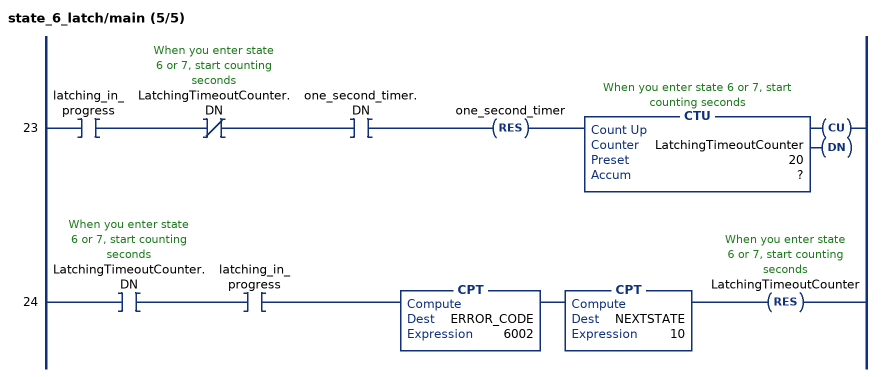
   23: XIC(latching_in_progress)XIO(LatchingTimeoutCounter.DN)XIC(one_second_timer.DN)RES(one_second_timer)CTU(LatchingTimeoutCounter,?,?);
   24: XIC(LatchingTimeoutCounter.DN)XIC(latching_in_progress)CPT(ERROR_CODE,6002)CPT(NEXTSTATE,10)RES(LatchingTimeoutCounter);
END_ROUTINE
END_PROGRAM
